// TIA Portal V18 export
FUNCTION "ER_lim_v_ws" : Void   // FC20, FBD
{ S7_Optimized_Access := 'TRUE' }
VERSION : 0.1
// stored: AutoNumber true, IsIECCheckEnabled false, SetENOAutomatically false, UDAEnableTagReadback false
   VAR_INPUT
      v_auto_USER : Real;
      v_absoluteMax_LOGIC : Real;
      v_fast_USER : Real;
      v_blind_USER : Real;
      v_crawl_LOGIC : Real;
   END_VAR
   VAR_OUTPUT
      ER_settings : Bool;
      wsER : WString;
   END_VAR
   VAR_TEMP
      tmp_fwdLEREV : Bool;
      tmp_fastL0 : Bool;
      tmp_fastLEslo : Bool;
      e_v_auto : Bool;
      e_v_blind : Bool;
      e_v_crawl : Bool;
      e_v_fast : Bool;
   END_VAR
BEGIN

REGION Network 1
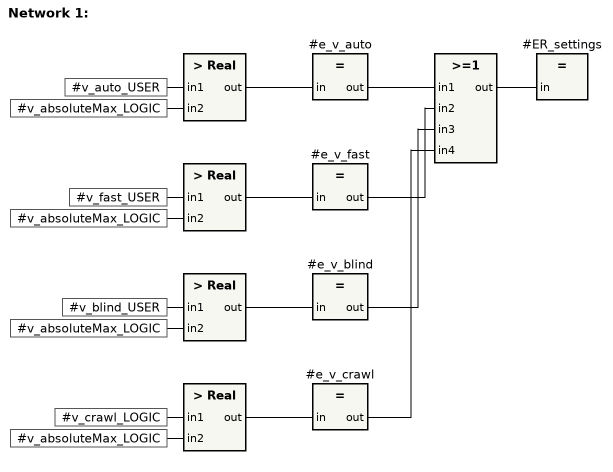
   #e_v_auto := #v_auto_USER > #v_absoluteMax_LOGIC;
   #e_v_fast := #v_fast_USER > #v_absoluteMax_LOGIC;
   #e_v_blind := #v_blind_USER > #v_absoluteMax_LOGIC;
   #e_v_crawl := #v_crawl_LOGIC > #v_absoluteMax_LOGIC;
   #ER_settings := #e_v_auto OR #e_v_fast OR #e_v_blind OR #e_v_crawl;
END_REGION

REGION Network 2 (SCL)
   IF #e_v_auto THEN
       #wsER := WSTRING#'v auto GT abs max';
   END_IF;
   IF #e_v_fast THEN
       #wsER := WSTRING#'v fast GT abs max';
   END_IF;
   IF #e_v_blind THEN
       #wsER := WSTRING#'v blind GT abs max';
   END_IF;
   IF #e_v_crawl THEN
       #wsER := WSTRING#'v crawl GT abs max';
   END_IF;
END_REGION
END_FUNCTION
